FUNCTION_BLOCK FB105
TITLE = 'pilot_Z4'
AUTHOR : CB

VAR
	pilot_Z4CONV1VAD : FB104;
END_VAR


BEGIN


NETWORK
TITLE =
//
//	pilot/pilot_Z4/pilot_Z4CONV1VAD
CALL #pilot_Z4CONV1VAD;




END_FUNCTION_BLOCK
